Fanuc KAREL source: ko00045.KL

-- PROVISIONAL review KL for V1013-1; original PC SHA256 8a6d36bd3a9d7a35f500c96006b36c603552dabe5d03e2a6ff872d90a3c2db7f
-- Incomplete behavior may be omitted. Consult companion uncertainty JSON. Do not deploy.
PROGRAM KO00045
%NOLOCKGROUP
BEGIN
  -- UNRESOLVED_PC offsets 5-12; opcodes 9D,23
  -- UNRESOLVED_PC offsets 17-69; opcodes 27,27,49,7E,AD,27,49,7E,AD,22,31,7E,4A
  -- UNRESOLVED_PC offsets 74-78; opcodes 7F
END KO00045
